// TIA Portal V19 export
TYPE "PPrf_SetUp"
// stored: Access Published
   STRUCT
      Aut : "PPrf_SetUp_Aut";
      Man : "PPrf_SetUp_Man";
   END_STRUCT;
END_TYPE
